FUNCTION_BLOCK ASR2_DELAY (* Delayed event propagation (ASR2 Adapter, Set und Reset je unabhaengig verzoegert) *)
  (* Standard: 61499-2; Description: Copyright (c) 2026 HR Agrartechnik GmbH This program and the accompanying materials are made available under the terms of the Eclipse Public License 2.0 which is available at https://www.eclipse.org/legal/epl-2.0/ SPDX-License-Identifier: EPL-2.0 *)
  (* Version 1.0, 2026-09-17, Franz Höpfinger, HR Agrartechnik GmbH, Wrapper fuer 2x E_DELAY ueber ASR2-Adapter - verzoegert SET und RESET eines Set/Reset-Kettenglieds (z.B. AX_T_FF_SR_SEQ) je um DT *)
  (* Version 1.1, 2026-09-17, Franz Höpfinger, HR Agrartechnik GmbH, Bugfix (Franz: 'ASR2_DELAY.fbt braucht 4 Zeiten', 'ATM waere hier richtig'): gemeinsamer Klartext-InputVar DT:TIME (nie ueber INIT initialisiert, UND SET/RESET faelschlich mit derselben Zeit) durch 2 getrennte ATM-Sockets DT_SET/DT_RESET ersetzt - SET- und RESET-Verzoegerung sind damit unabhaengig voneinander einstellbar UND sauber ueber initval_ATM+INIT/INITO initialisierbar. *)
  (* Version 1.2, 2026-09-17, Franz Höpfinger, HR Agrartechnik GmbH, Bugfix (Franz: 'ASR2_DELAY.fbt braucht 4 Zeiten und 4 STOP', analog zur AE2_DELAY-Korrektur): ASR2 ist wie AE2 echt bidirektional (EI_SET/EI_RESET/EO_SET/EO_RESET je Socket UND Plug) - bisher wurde nur die Vorwaerts-Richtung verzoegert. Jetzt 4 unabhaengige E_DELAY-Instanzen (SET/RESET x Vorwaerts/Rueckwaerts), 4 ATM-Zeiten PT_SET_FWD/PT_SET_BWD/PT_RESET_FWD/PT_RESET_BWD (vormals DT_SET/DT_RESET, DT-Praefix wegen 'DT is a reserved keyword' auf PT umbenannt) und 4 AE-Stop-Sockets STOP_SET_FWD/STOP_SET_BWD/STOP_RESET_FWD/STOP_RESET_BWD. *)
  PACKAGE adapter::events::bidirectional;
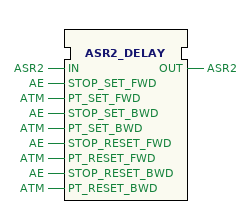
  SOCKETS
    IN : adapter::types::bidirectional::ASR2; (* Set/Reset vom vorherigen Kettenglied (bidirektional: Vorwaerts herein, Rueckwaerts hinaus) *)
    STOP_SET_FWD : adapter::types::unidirectional::AE; (* Stop delay SET Vorwaerts *)
    PT_SET_FWD : adapter::types::unidirectional::ATM; (* Preset Time SET Vorwaerts (IN.EO_SET->OUT.EO_SET) *)
    STOP_SET_BWD : adapter::types::unidirectional::AE; (* Stop delay SET Rueckwaerts *)
    PT_SET_BWD : adapter::types::unidirectional::ATM; (* Preset Time SET Rueckwaerts (OUT.EI_SET->IN.EI_SET) *)
    STOP_RESET_FWD : adapter::types::unidirectional::AE; (* Stop delay RESET Vorwaerts *)
    PT_RESET_FWD : adapter::types::unidirectional::ATM; (* Preset Time RESET Vorwaerts (IN.EO_RESET->OUT.EO_RESET) *)
    STOP_RESET_BWD : adapter::types::unidirectional::AE; (* Stop delay RESET Rueckwaerts *)
    PT_RESET_BWD : adapter::types::unidirectional::ATM; (* Preset Time RESET Rueckwaerts (OUT.EI_RESET->IN.EI_RESET) *)
  END_SOCKETS
  PLUGS
    OUT : adapter::types::bidirectional::ASR2; (* Verzoegertes Set/Reset, an naechstes Kettenglied (bidirektional: Vorwaerts hinaus, Rueckwaerts herein) *)
  END_PLUGS
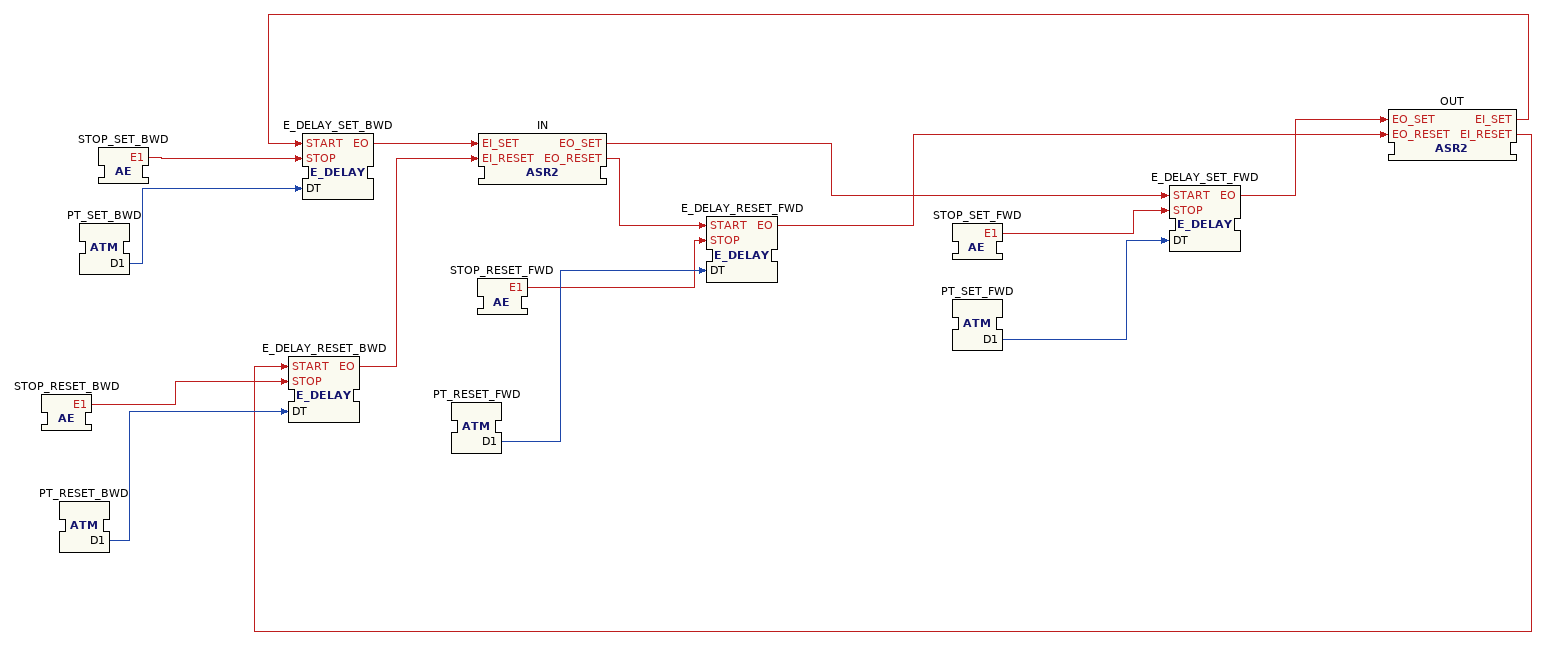
  FBS
    E_DELAY_SET_FWD : iec61499::events::E_DELAY;
    E_DELAY_SET_BWD : iec61499::events::E_DELAY;
    E_DELAY_RESET_FWD : iec61499::events::E_DELAY;
    E_DELAY_RESET_BWD : iec61499::events::E_DELAY;
  END_FBS
  EVENT_CONNECTIONS
    IN.EO_SET TO E_DELAY_SET_FWD.START;
    STOP_SET_FWD.E1 TO E_DELAY_SET_FWD.STOP;
    E_DELAY_SET_FWD.EO TO OUT.EO_SET;
    OUT.EI_SET TO E_DELAY_SET_BWD.START;
    STOP_SET_BWD.E1 TO E_DELAY_SET_BWD.STOP;
    E_DELAY_SET_BWD.EO TO IN.EI_SET;
    IN.EO_RESET TO E_DELAY_RESET_FWD.START;
    STOP_RESET_FWD.E1 TO E_DELAY_RESET_FWD.STOP;
    E_DELAY_RESET_FWD.EO TO OUT.EO_RESET;
    OUT.EI_RESET TO E_DELAY_RESET_BWD.START;
    STOP_RESET_BWD.E1 TO E_DELAY_RESET_BWD.STOP;
    E_DELAY_RESET_BWD.EO TO IN.EI_RESET;
  END_CONNECTIONS
  DATA_CONNECTIONS
    PT_SET_FWD.D1 TO E_DELAY_SET_FWD.DT;
    PT_SET_BWD.D1 TO E_DELAY_SET_BWD.DT;
    PT_RESET_FWD.D1 TO E_DELAY_RESET_FWD.DT;
    PT_RESET_BWD.D1 TO E_DELAY_RESET_BWD.DT;
  END_CONNECTIONS
END_FUNCTION_BLOCK
